FUNCTION_BLOCK SET_SPINDLE_DATA (* Sets data to activate/deactivate machine spindle *)
  (* Standard: 61499-2 *)
  (* Version 1.0, 18-04-2012, GASR, Universidade do Estado de Santa Catarina *)
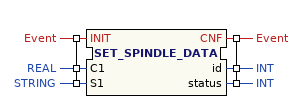
  EVENT_INPUT
    INIT WITH C1, S1;
  END_EVENT
  EVENT_OUTPUT
    CNF WITH id, status;
  END_EVENT
  VAR_INPUT
    C1 : REAL; (* Coeficient 1 *)
    S1 : STRING; (* String 1 *)
  END_VAR
  VAR_OUTPUT
    id : INT;
    status : INT;
  END_VAR
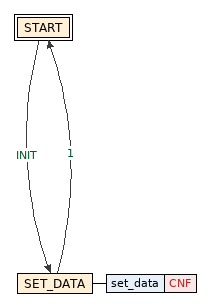
  EC_STATES
    START;
    SET_DATA : set_data -> CNF;
  END_STATES
  EC_TRANSITIONS
    START TO SET_DATA := INIT;
    SET_DATA TO START := 1;
  END_TRANSITIONS
  ALGORITHM set_data IN Lua:
id = C1
if( S1 == "on" ) then
    status = 1
else
    status = 0
end
  END_ALGORITHM
END_FUNCTION_BLOCK
